// TIA Portal V16 export
// export: Created 2025-08-01T13:38:03.4500506Z, ExportSetting WithDefaults, DisplayName Totally Integrated Automation Portal, DisplayVersion V16, DisplayName TIA Portal Version Control Interface, DisplayVersion V16, DisplayName TIA Portal Openness, DisplayVersion V16, DisplayName STEP 7 Professional, DisplayVersion V16, DisplayName STEP 7 Safety, DisplayVersion V16, DisplayName WinCC Advanced, DisplayVersion V16
DATA_BLOCK "BlowOff_Timer_ManualDB"   // DB83
VERSION : 0.1
// stored: AutoNumber true, InstanceOfName BlowOff_Timer, InstanceOfType FB
"BlowOff_Timer"
   // VAR_INPUT
   //    Enable : Bool;
   //    CycleTime : Time;
   //    PulseDuration : Time;
   //    NowTime : Time;
   // END_VAR
   // VAR_OUTPUT
   //    Q_Pulse : Bool;
   // END_VAR
   // VAR RETAIN
   //    CycleTimer : TON;
   //    PulseTimer : TON;
   //    State { S7_SetPoint := 'True'} : Int;
   //    S_PEXT : Int;
   // END_VAR
BEGIN
END_DATA_BLOCK
